(* PLC project PLC1, Beckhoff Automation GmbH TwinCAT PLC Control 3.5.13.21 *)
(* stored: creationDateTime 2022-08-11T18:55:06.8051548, modificationDateTime 2022-08-11T18:55:06.8051548 *)

FUNCTION_BLOCK FB_Word_To_Bool
VAR_INPUT
	inWord : WORD;
END_VAR
VAR_OUTPUT
	outArrayOfBool : ARRAY [0..15] OF BOOL;
END_VAR
VAR
END_VAR

            outArrayOfBool[0] := inWord.0;
outArrayOfBool[1] := inWord.1;
outArrayOfBool[2] := inWord.2;
outArrayOfBool[3] := inWord.3;
outArrayOfBool[4] := inWord.4;
outArrayOfBool[5] := inWord.5;
outArrayOfBool[6] := inWord.6;
outArrayOfBool[7] := inWord.7;
outArrayOfBool[8] := inWord.8;
outArrayOfBool[9] := inWord.9;
outArrayOfBool[10] := inWord.10;
outArrayOfBool[11] := inWord.11;
outArrayOfBool[12] := inWord.12;
outArrayOfBool[13] := inWord.13;
outArrayOfBool[14] := inWord.14;
outArrayOfBool[15] := inWord.15;
          
END_FUNCTION_BLOCK
